GLOBALCONSTANTS EmergencyStopDiagCodes (* PLCopen Safety Part 1 Ch. 6.5.6 - SF_EmergencyStop-specific DiagCode values *)
  (* Standard: 61499-1; Description: Copyright (c) 2026 Meisterschulen am Ostbahnhof This program and the accompanying materials are made available under the terms of the Eclipse Public License 2.0 which is available at https://www.eclipse.org/legal/epl-2.0/ SPDX-License-Identifier: EPL-2.0 *)
  (* Version 1.0, 2026-10-09, Franz Höpfinger, Meisterschulen am Ostbahnhof, Source: PLCopen TC5 Safety Part 1, Version 2.10, Chapter 6.5.6 DiagCode table. See also DiagCodes.gcf for the shared IDLE code. *)
  PACKAGE logiBUS::safety::PLCopen::const;
  VAR_GLOBAL CONSTANT
    INIT : WORD := 16#8001; (* 8001 - activated, checking S_StartReset *)
    WAIT_ESTOP_IN_1 : WORD := 16#8802; (* 8802 - first activation, waiting for S_EStopIn *)
    WAIT_RESET_1 : WORD := 16#8402; (* 8402 - first activation, waiting for Reset edge *)
    WAIT_ESTOP_IN_2 : WORD := 16#8804; (* 8804 - safety demand detected, waiting for S_EStopIn *)
    WAIT_RESET_2 : WORD := 16#8404; (* 8404 - waiting for S_AutoReset or Reset edge *)
    SAFETY_OUTPUT_ENABLED : WORD := 16#8000; (* 8000 - S_EStopOut is TRUE *)
    RESET_ERROR_1 : WORD := 16#C001; (* C001 - Reset stuck TRUE while waiting for S_EStopIn (1st) *)
    RESET_ERROR_2 : WORD := 16#C011; (* C011 - Reset stuck TRUE while waiting for S_EStopIn (2nd) *)
  END_VAR
END_GLOBALCONSTANTS
